RoboDK station: Stringer B-Corner-Top-Short-BOX2.rdk

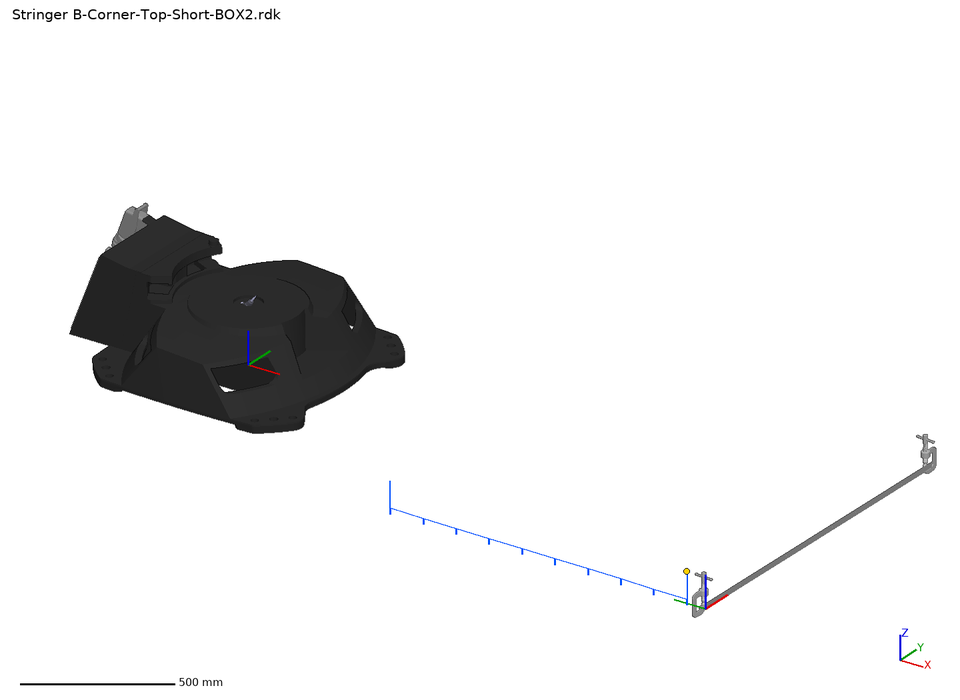
[picture v0: the station drawn from its stored meshes, robots at their saved joint values, targets as dots, program paths as lines]
Station Stringer B-Corner-Top-Short-BOX2 (saved by RoboDK 5.2.3). Poses are relative to the parent item; angles as X-Y-Z fixed-axis rotations.
  - frame KUKA KR 210 R2700 extra Base at (0, 0, 0) mm
    - robot KUKA KR 210 R2700 extra: 6 axes, payload 210 kg, reach 2696 mm, repeatability 0.06 mm, weight 1068 kg
        joint limits [-185, -140, -120, -350, -125, -350] to [185, -5, 155, 350, 125, 350]; home [0, -90, 90, 0, 0, 0]; saved at [-39.14, -26.646, 86.085, 93.624, 23.455, -126.261]
      - tool Spindle, TCP at (32, 0, 260) mm, rotated rx 0 ry 39 rz 0 deg, size 157.3 x 72 x 259.9 mm
  - frame Frame 2 at (1800, 0, -372.68) mm, rotated rx 0 ry 0 rz 90 deg
    - object Stringer B-Corner-Top-Short-BOX2 at (0, 0, 0) mm, rotated rx 0 ry 0 rz -90 deg, 10 curves, geometry from Point 10
    - object L-Stringer B-top-corner-short - box2 at (0, 0, 0) mm, size 1281.1 x 20 x 20 mm, 1 curves, geometry from L-Stringer B-top-corner-short - box2.stl
  - machining project Point settings: rotZ(0) | rotX(0)*rotY(0) | rotz(0) | onStart | onPathStart | onApproach | onPoint | onRetract | onFinish | SetRPM(%1) | SetTool(%1) | Extruder(%1) | default | default | OutOnMov(%1) | OutOffMov(%1) | onPathFinish | M_RunCode(%1)
  - program Point (61 instructions, listed below)
  - object FinalClamp at (1786.94, 1254.06, -310.13) mm, rotated rx 128.54 ry 87.64 rz 128.37 deg, size 145.3 x 71.1 x 72 mm, geometry from FinalClamp.stp
  - object FinalClamp2 at (1782.58, 13.73, -311.49) mm, rotated rx 138.93 ry 89.04 rz -45.11 deg, size 145.3 x 71.1 x 72 mm, geometry from FinalClamp.stp
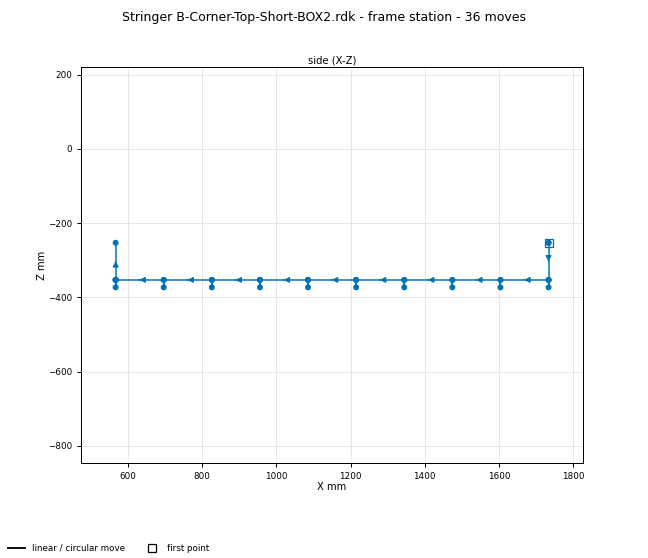
[picture p0: tool path of Stringer B-Corner-Top-Short-BOX2.rdk in frame station, 36 of 36 moves have a stored position in this frame; points joined in program order, loops and branches not executed]

--- program Point (robot KUKA KR 210 R2700 extra) ---
  Smooth(1)
  Set speed (1000.0 mm/s)
  Set Ref.: Frame 2
  Set Tool: Spindle
  Show Spindle
  MoveJ 1 to (-11.4, 66.57, 120) mm, rotated rx 180 ry 0 rz 180 deg; joints [-2.517, -34.014, 111.85, 176.493, 26.853, -178.826]
  MoveL 2 to (-11.4, 66.57, 120) mm, rotated rx 180 ry 0 rz 180 deg; joints [-2.517, -34.014, 111.85, 176.493, 26.853, -178.826]
  MoveL 3 to (-11.4, 66.57, 20) mm, rotated rx 180 ry 0 rz -180 deg; joints [-2.517, -28.684, 109.207, 176.786, 29.535, -179.16]
  MoveL 4 to (-11.4, 66.57, 20) mm, rotated rx 180 ry 0 rz -180 deg; joints [-2.517, -28.684, 109.207, 176.786, 29.535, -179.16]
  Set speed (50.0 mm/s)
  MoveL 5 to (-11.4, 66.57, 0) mm, rotated rx -180 ry 0 rz -180 deg; joints [-2.517, -27.626, 108.632, 176.833, 30.016, -179.214]
  MoveL 6 to (-11.4, 66.57, 20) mm, rotated rx 180 ry 0 rz -180 deg; joints [-2.517, -28.684, 109.207, 176.786, 29.535, -179.16]
  Set speed (1000.0 mm/s)
  MoveL 7 to (-11.4, 196.13, 20) mm, rotated rx -180 ry 0 rz 180 deg; joints [-7.379, -28.603, 108.626, 170.443, 29.129, -177.38]
  Set speed (50.0 mm/s)
  MoveL 8 to (-11.4, 196.13, 0) mm, rotated rx -180 ry 0 rz -180 deg; joints [-7.379, -27.551, 108.052, 170.583, 29.601, -177.541]
  MoveL 9 to (-11.4, 196.13, 20) mm, rotated rx -180 ry 0 rz 180 deg; joints [-7.379, -28.603, 108.626, 170.443, 29.129, -177.38]
  Set speed (1000.0 mm/s)
  MoveL 10 to (-11.4, 325.68, 20) mm, rotated rx 180 ry 0 rz 180 deg; joints [-12.136, -28.431, 107.473, 163.831, 28.366, -175.175]
  Set speed (50.0 mm/s)
  MoveL 11 to (-11.4, 325.68, 0) mm, rotated rx -180 ry 0 rz 180 deg; joints [-12.136, -27.388, 106.903, 164.071, 28.82, -175.448]
  MoveL 12 to (-11.4, 325.68, 20) mm, rotated rx 180 ry 0 rz 180 deg; joints [-12.136, -28.431, 107.473, 163.831, 28.366, -175.175]
  Set speed (1000.0 mm/s)
  MoveL 13 to (-11.4, 455.24, 20) mm, rotated rx -180 ry 0 rz -180 deg; joints [-16.73, -28.144, 105.753, 156.762, 27.331, -172.268]
  Set speed (50.0 mm/s)
  MoveL 14 to (-11.4, 455.24, 0) mm, rotated rx 180 ry 0 rz 180 deg; joints [-16.73, -27.116, 105.189, 157.11, 27.758, -172.661]
  MoveL 15 to (-11.4, 455.24, 20) mm, rotated rx -180 ry 0 rz -180 deg; joints [-16.73, -28.144, 105.753, 156.762, 27.331, -172.268]
  Set speed (1000.0 mm/s)
  MoveL 16 to (-11.4, 584.79, 20) mm, rotated rx -180 ry 0 rz -180 deg; joints [-21.112, -27.714, 103.474, 149.041, 26.145, -168.4]
  Set speed (50.0 mm/s)
  MoveL 17 to (-11.4, 584.79, 0) mm, rotated rx 180 ry 0 rz 180 deg; joints [-21.112, -26.704, 102.916, 149.507, 26.534, -168.921]
  MoveL 18 to (-11.4, 584.79, 20) mm, rotated rx -180 ry 0 rz -180 deg; joints [-21.112, -27.714, 103.474, 149.041, 26.145, -168.4]
  Set speed (1000.0 mm/s)
  MoveL 19 to (-11.4, 714.35, 20) mm, rotated rx -180 ry 0 rz -180 deg; joints [-25.251, -27.107, 100.638, 140.487, 24.957, -163.345]
  Set speed (50.0 mm/s)
  MoveL 20 to (-11.4, 714.35, 0) mm, rotated rx 180 ry 0 rz 180 deg; joints [-25.251, -26.118, 100.087, 141.077, 25.296, -163.996]
  MoveL 21 to (-11.4, 714.35, 20) mm, rotated rx -180 ry 0 rz -180 deg; joints [-25.251, -27.107, 100.638, 140.487, 24.957, -163.345]
  Set speed (1000.0 mm/s)
  MoveL 22 to (-11.4, 843.91, 20) mm, rotated rx -180 ry 0 rz -180 deg; joints [-29.127, -26.288, 97.248, 130.984, 23.94, -156.963]
  Set speed (50.0 mm/s)
  MoveL 23 to (-11.4, 843.91, 0) mm, rotated rx -180 ry 0 rz -180 deg; joints [-29.127, -25.323, 96.703, 131.691, 24.218, -157.737]
  MoveL 24 to (-11.4, 843.91, 20) mm, rotated rx -180 ry 0 rz -180 deg; joints [-29.127, -26.288, 97.248, 130.984, 23.94, -156.963]
  Set speed (1000.0 mm/s)
  MoveL 25 to (-11.4, 973.46, 20) mm, rotated rx 180 ry 0 rz 180 deg; joints [-32.731, -25.225, 93.299, 120.558, 23.275, -149.272]
  Set speed (50.0 mm/s)
  MoveL 26 to (-11.4, 973.46, 0) mm, rotated rx -180 ry 0 rz -180 deg; joints [-32.731, -24.284, 92.758, 121.354, 23.482, -150.139]
  MoveL 27 to (-11.4, 973.46, 20) mm, rotated rx 180 ry 0 rz 180 deg; joints [-32.731, -25.225, 93.299, 120.558, 23.275, -149.272]
  Set speed (1000.0 mm/s)
  MoveL 28 to (-11.4, 1103.02, 20) mm, rotated rx -180 ry 0 rz -180 deg; joints [-36.065, -23.883, 88.773, 109.453, 23.136, -140.52]
  Set speed (50.0 mm/s)
  MoveL 29 to (-11.4, 1103.02, 0) mm, rotated rx 180 ry 0 rz 180 deg; joints [-36.065, -22.965, 88.235, 110.285, 23.265, -141.426]
  MoveL 30 to (-11.4, 1103.02, 20) mm, rotated rx -180 ry 0 rz -180 deg; joints [-36.065, -23.883, 88.773, 109.453, 23.136, -140.52]
  Set speed (1000.0 mm/s)
  MoveL 31 to (-11.4, 1232.57, 20) mm, rotated rx -180 ry 0 rz -180 deg; joints [-39.14, -22.224, 83.64, 98.136, 23.658, -131.183]
  Set speed (50.0 mm/s)
  MoveL 32 to (-11.4, 1232.57, 0) mm, rotated rx 180 ry 0 rz 180 deg; joints [-39.14, -21.329, 83.1, 98.937, 23.711, -132.058]
  MoveL 33 to (-11.4, 1232.57, 20) mm, rotated rx -180 ry 0 rz -180 deg; joints [-39.14, -22.224, 83.64, 98.136, 23.658, -131.183]
  MoveL 34 to (-11.4, 1232.57, 20) mm, rotated rx -180 ry 0 rz -180 deg; joints [-39.14, -22.224, 83.64, 98.136, 23.658, -131.183]
  Set speed (1000.0 mm/s)
  MoveL 35 to (-11.4, 1232.57, 20) mm, rotated rx -180 ry 0 rz -180 deg; joints [-39.14, -22.224, 83.64, 98.136, 23.658, -131.183]
  MoveL 36 to (-11.4, 1232.57, 120) mm, rotated rx -180 ry 0 rz -180 deg; joints [-39.14, -26.646, 86.085, 93.624, 23.455, -126.261]
